              Wait Sleep waitTime=0.3
              If barrenoActual≟13
                MoveDirectionNode (selectedDirection=ZPlus toolParams=0.03, 0.04)
                  Until DISTANCE (allowActions=false deceleration=3 distanceNodeType=STOP) Distance=0.03; motionParameters(blendRadius=0)
                MoveJ speed 60 deg/s, acceleration 80 deg/s^2 (useActiveTCP=true) feature=Base
                  Waypoint Zona_der1: TCP in base x=-721.714 y=-174.597 z=506.289 mm, rx=2.1128 ry=-2.325 rz=0 rad; joints [0.057, -90.231, 90.368, -0.664, 90.292, 0.009] deg
                  Waypoint Posicion_Cero: TCP in base x=0.641 y=-324.742 z=1651.532 mm, rx=-0.0042 ry=-0.0154 rz=-3.0499 rad; joints [-0.001, -90.003, -0.001, -90, 0, 0.002] deg
                Call Quitar_Broca_Chida
                Call Poner_Broca
                MoveJ speed 60 deg/s, acceleration 80 deg/s^2 (useActiveTCP=true) feature=Base
                  Waypoint Posicion_Cero: TCP in base x=0.641 y=-324.742 z=1651.532 mm, rx=-0.0042 ry=-0.0154 rz=-3.0499 rad; joints [-0.001, -90.003, -0.001, -90, 0, 0.002] deg
                  Waypoint Zona_der1: TCP in base x=-721.714 y=-174.597 z=506.289 mm, rx=2.1128 ry=-2.325 rz=0 rad; joints [0.057, -90.231, 90.368, -0.664, 90.292, 0.009] deg
              ElseIf barrenoActual≟27
                MoveDirectionNode (selectedDirection=ZPlus toolParams=0.03, 0.04)
                  Until DISTANCE (allowActions=false deceleration=3 distanceNodeType=STOP) Distance=0.03; motionParameters(blendRadius=0)
                MoveJ speed 60 deg/s, acceleration 80 deg/s^2 (useActiveTCP=true) feature=Base
                  Waypoint Zona_der1: TCP in base x=-721.714 y=-174.597 z=506.289 mm, rx=2.1128 ry=-2.325 rz=0 rad; joints [0.057, -90.231, 90.368, -0.664, 90.292, 0.009] deg
                  Waypoint Posicion_Cero: TCP in base x=0.641 y=-324.742 z=1651.532 mm, rx=-0.0042 ry=-0.0154 rz=-3.0499 rad; joints [-0.001, -90.003, -0.001, -90, 0, 0.002] deg
                Call Quitar_Broca_Chida
                Set DigitalOutput pin=carrusel_home; digitalValue=1
                Wait Sleep waitTime=1
                Set DigitalOutput pin=carrusel_home; digitalValue=0
                Set ExpressionOutput pin=mensaje_mw10; expression=85
                Wait DigitalInput pin=Continuar_M30; digitalValue=1
                Wait Sleep waitTime=1
                Set ExpressionOutput pin=mensaje_mw10; expression=120
                Wait DigitalInput pin=Continuar_M30; digitalValue=1
                Wait Sleep waitTime=1
                Set DigitalOutput pin=carrusel_home; digitalValue=1
                Wait Sleep waitTime=1
                Set DigitalOutput pin=carrusel_home; digitalValue=0
                Set ExpressionOutput pin=mensaje_mw10; expression=90
                Wait DigitalInput pin=Continuar_M30; digitalValue=1
                Wait Sleep waitTime=1
                Call Poner_Broca
                broca := 217
                MoveJ speed 60 deg/s, acceleration 80 deg/s^2 (useActiveTCP=true) feature=Base
                  Waypoint Posicion_Cero: TCP in base x=0.641 y=-324.742 z=1651.532 mm, rx=-0.0042 ry=-0.0154 rz=-3.0499 rad; joints [-0.001, -90.003, -0.001, -90, 0, 0.002] deg
                  Waypoint Zona_der1: TCP in base x=-721.714 y=-174.597 z=506.289 mm, rx=2.1128 ry=-2.325 rz=0 rad; joints [0.057, -90.231, 90.368, -0.664, 90.292, 0.009] deg
                Set ExpressionOutput pin=mensaje_mw10; expression=95
                Wait DigitalInput pin=Continuar_M30; digitalValue=1
                Wait Sleep waitTime=1
                Set ExpressionOutput pin=mensaje_mw10; expression=150
                Wait DigitalInput pin=Continuar_M30; digitalValue=1
                Wait Sleep waitTime=1
              barrenoActual := barrenoActual+1
        Folder Linea 1 a 217
          broca := 217
          Folder Buje_inicial
            Buje_Inicial := L1B2
          Folder Buje_final
            Buje_Final := L1B1
          barrenosTotales := 27
          barrenoActual := 1
          Loop While (checkContinuously=false) expression=barrenoActual≤barrenosTotales
            MoveL speed 250 mm/s, acceleration 1200 mm/s^2 (useActiveTCP=true) feature=Base
              bajada_broca := p[0,0,0.018,0,0,0]
              internos := interpolate_pose(Buje_Inicial, Buje_Final, ((barrenoActual)-1)/((barrenosTotales)-1))
              Wait Sleep waitTime=2
              Folder Alturas
                If barrenoActual≟1 or barrenoActual≟3 or barrenoActual≟5 or barrenoActual≟7 or barrenoActual≟9 or barrenoActual≟11 or barrenoActual≟13 or barrenoActual≟15 or barrenoActual≟17 or barrenoActual≟19 or barrenoActual≟21 or barrenoActual≟23 or barrenoActual≟25 or barrenoActual≟27
                  Set ExpressionOutput pin=mensaje_mw10; expression=200
                  Wait DigitalInput pin=Continuar_M30; digitalValue=1
                  Wait Sleep waitTime=1
                  Set ExpressionOutput pin=mensaje_mw10; expression=150
                  Wait Sleep waitTime=1
                MoveJ speed 30 deg/s, acceleration 40 deg/s^2 (useActiveTCP=true) feature=Base
                  Waypoint Waypoint (Variable): variable=internos
                Wait Sleep waitTime=2
                If P1h[2]<P2h[2]
                  acomodo := (altura/(barrenosTotales-1))*(barrenoActual-1)
                  tcp := get_actual_tcp_pose()
                  offset_altura := p[tcp[0],tcp[1],((alta-0.0095)-(acomodo/1000)),tcp[3],tcp[4],tcp[5]]
                  MoveL speed 250 mm/s, acceleration 1200 mm/s^2 (useActiveTCP=true) feature=Base
                    Waypoint Waypoint (Variable): motionParameters(jointSpeed=1.047198 jointAcceleration=1.396263 cartesianSpeed=0.03 cartesianAcceleration=0.04); variable=offset_altura
                Else 
                  acomodo := (altura/(barrenosTotales-1))*(26-(barrenoActual-1))
                  tcp := get_actual_tcp_pose()
                  offset_altura := p[tcp[0],tcp[1],((alta-0.0095)-(acomodo/1000)),tcp[3],tcp[4],tcp[5]]
                  MoveL speed 250 mm/s, acceleration 1200 mm/s^2 (useActiveTCP=true) feature=Base
                    Waypoint Waypoint (Variable): motionParameters(jointSpeed=1.047198 jointAcceleration=1.396263 cartesianSpeed=0.03 cartesianAcceleration=0.04); variable=offset_altura
              Folder Freemove
                Wait Sleep waitTime=2
                Script: freedrive_mode()
                Wait Sleep waitTime=2.5
                Script: end_freedrive_mode()
              Wait Sleep waitTime=0.3
              Set DigitalOutput pin=config_out[1]; digitalValue=1
              Wait Sleep waitTime=1
              Wait Sleep waitTime=0.3
              Wait Sleep waitTime=0.3
              Wait Sleep waitTime=0.3
              Loop Counting (count=1) loopVariable(name=Loop_56)
                Poses_taladrado := pose_sub(get_actual_tcp_pose(), bajada_broca)
                Waypoint Waypoint (Variable): motionParameters(jointSpeed=1.047198 jointAcceleration=1.396263 cartesianSpeed=0.001 cartesianAcceleration=0.005); variable=Poses_taladrado
                If bajada_broca≟p[0,0,0.018,0,0,0]
                  num_barreno := str_cat("Barreno: ",barrenoActual)
                  tcp_actual := get_actual_tcp_pose()
                  X_actual := str_cat("     X: ",tcp_actual[0])
                  Y_actual := str_cat("     Y: ",tcp_actual[1])
                  pos_barreno := str_cat(X_actual,Y_actual)
                  Script: textmsg(num_barreno,pos_barreno)
                Poses_taladrado := pose_add(get_actual_tcp_pose(), bajada_broca)
                Waypoint Waypoint (Variable): motionParameters(jointSpeed=1.047198 jointAcceleration=1.396263 cartesianSpeed=0.01 cartesianAcceleration=0.01); variable=Poses_taladrado
                bajada_broca := pose_add(bajada_broca, p[0,0,0.018,0,0,0])
              MoveDirectionNode (selectedDirection=ZPlus toolParams=0.01, 0.01)
                Until DISTANCE (allowActions=false deceleration=3 distanceNodeType=STOP) Distance=0.05; motionParameters(blendRadius=0)
              MoveJ speed 30 deg/s, acceleration 40 deg/s^2 (useActiveTCP=true) feature=Base
                Waypoint Waypoint (Variable): variable=internos
              Wait Sleep waitTime=0.3
              Set DigitalOutput pin=config_out[1]; digitalValue=0
              Wait Sleep waitTime=0.3
              If barrenoActual≟13 or barrenoActual≟27
                MoveDirectionNode (selectedDirection=ZPlus toolParams=0.04, 0.03)
                  Until DISTANCE (allowActions=false deceleration=3 distanceNodeType=STOP) Distance=0.03; motionParameters(blendRadius=0)
                MoveJ speed 30 deg/s, acceleration 40 deg/s^2 (useActiveTCP=true) feature=Base
                  Waypoint Zona_der1: TCP in base x=-721.714 y=-174.597 z=506.289 mm, rx=2.1128 ry=-2.325 rz=0 rad; joints [0.057, -90.231, 90.368, -0.664, 90.292, 0.009] deg
                  Waypoint Posicion_Cero: TCP in base x=0.641 y=-324.742 z=1651.532 mm, rx=-0.0042 ry=-0.0154 rz=-3.0499 rad; joints [-0.001, -90.003, -0.001, -90, 0, 0.002] deg
                Call Quitar_Broca_Chida
                If barrenoActual≟13
                  Call Poner_Broca
                ElseIf barrenoActual≟27
                  Call Poner_Broca
                MoveJ speed 30 deg/s, acceleration 40 deg/s^2 (useActiveTCP=true) feature=Base
                  Waypoint Posicion_Cero: TCP in base x=0.641 y=-324.742 z=1651.532 mm, rx=-0.0042 ry=-0.0154 rz=-3.0499 rad; joints [-0.001, -90.003, -0.001, -90, 0, 0.002] deg
                  Waypoint Zona_der1: TCP in base x=-721.714 y=-174.597 z=506.289 mm, rx=2.1128 ry=-2.325 rz=0 rad; joints [0.057, -90.231, 90.368, -0.664, 90.292, 0.009] deg
              barrenoActual := barrenoActual+1
        Folder Linea 2 a 217
          broca := 217
          Folder Buje_inicial
            Buje_Inicial := L2B2
          Folder Buje_final
            Buje_Final := L2B1
          barrenosTotales := 27
          barrenoActual := 1
          Loop While (checkContinuously=false) expression=barrenoActual≤barrenosTotales
            MoveL speed 250 mm/s, acceleration 1200 mm/s^2 (useActiveTCP=true) feature=Base
              bajada_broca := p[0,0,0.018,0,0,0]
              internos := interpolate_pose(Buje_Inicial, Buje_Final, ((barrenoActual)-1)/((barrenosTotales)-1))
              Folder Alturas
                If barrenoActual≟1 or barrenoActual≟3 or barrenoActual≟5 or barrenoActual≟7 or barrenoActual≟9 or barrenoActual≟11 or barrenoActual≟13 or barrenoActual≟15 or barrenoActual≟17 or barrenoActual≟19 or barrenoActual≟21 or barrenoActual≟23 or barrenoActual≟25 or barrenoActual≟27
                  Set ExpressionOutput pin=mensaje_mw10; expression=200
                  Wait DigitalInput pin=Continuar_M30; digitalValue=1
                  Wait Sleep waitTime=1
                  Set ExpressionOutput pin=mensaje_mw10; expression=150
                  Wait Sleep waitTime=1
                MoveJ speed 30 deg/s, acceleration 40 deg/s^2 (useActiveTCP=true) feature=Base
                  Waypoint Waypoint (Variable): variable=internos
                Wait Sleep waitTime=2
                If P1h[2]<P2h[2]
                  acomodo := (altura/(barrenosTotales-1))*(barrenoActual-1)
                  tcp := get_actual_tcp_pose()
                  offset_altura := p[tcp[0],tcp[1],((alta-0.0095)-(acomodo/1000)),tcp[3],tcp[4],tcp[5]]
                  MoveL speed 250 mm/s, acceleration 1200 mm/s^2 (useActiveTCP=true) feature=Base
                    Waypoint Waypoint (Variable): motionParameters(jointSpeed=1.047198 jointAcceleration=1.396263 cartesianSpeed=0.03 cartesianAcceleration=0.04); variable=offset_altura
                Else 
                  acomodo := (altura/(barrenosTotales-1))*(26-(barrenoActual-1))
                  tcp := get_actual_tcp_pose()
                  offset_altura := p[tcp[0],tcp[1],((alta-0.0095)-(acomodo/1000)),tcp[3],tcp[4],tcp[5]]
                  MoveL speed 250 mm/s, acceleration 1200 mm/s^2 (useActiveTCP=true) feature=Base
                    Waypoint Waypoint (Variable): motionParameters(jointSpeed=1.047198 jointAcceleration=1.396263 cartesianSpeed=0.03 cartesianAcceleration=0.04); variable=offset_altura
              Folder Freemove
                Wait Sleep waitTime=2
                Script: freedrive_mode()
                Wait Sleep waitTime=2.5
                Script: end_freedrive_mode()
              Wait Sleep waitTime=0.3
              Set DigitalOutput pin=config_out[1]; digitalValue=1
              Wait Sleep waitTime=1
              Wait Sleep waitTime=0.3
              Wait Sleep waitTime=0.3
              Wait Sleep waitTime=0.3
              Loop Counting (count=1) loopVariable(name=Loop_58)
                Poses_taladrado := pose_sub(get_actual_tcp_pose(), bajada_broca)
                Waypoint Waypoint (Variable): motionParameters(jointSpeed=1.047198 jointAcceleration=1.396263 cartesianSpeed=0.001 cartesianAcceleration=0.005); variable=Poses_taladrado
                If bajada_broca≟p[0,0,0.018,0,0,0]
                  num_barreno := str_cat("Barreno: ",barrenoActual)
                  tcp_actual := get_actual_tcp_pose()
                  X_actual := str_cat("     X: ",tcp_actual[0])
                  Y_actual := str_cat("     Y: ",tcp_actual[1])
                  pos_barreno := str_cat(X_actual,Y_actual)
                  Script: textmsg(num_barreno,pos_barreno)
                Poses_taladrado := pose_add(get_actual_tcp_pose(), bajada_broca)
                Waypoint Waypoint (Variable): motionParameters(jointSpeed=1.047198 jointAcceleration=1.396263 cartesianSpeed=0.01 cartesianAcceleration=0.01); variable=Poses_taladrado
                bajada_broca := pose_add(bajada_broca, p[0,0,0.018,0,0,0])
              MoveDirectionNode (selectedDirection=ZPlus toolParams=0.01, 0.01)
                Until DISTANCE (allowActions=false deceleration=3 distanceNodeType=STOP) Distance=0.05; motionParameters(blendRadius=0)
              MoveJ speed 30 deg/s, acceleration 40 deg/s^2 (useActiveTCP=true) feature=Base
                Waypoint Waypoint (Variable): variable=internos
              Wait Sleep waitTime=0.3
              Set DigitalOutput pin=config_out[1]; digitalValue=0
              Wait Sleep waitTime=0.3
              If barrenoActual≟13
                MoveDirectionNode (selectedDirection=ZPlus toolParams=0.03, 0.04)
                  Until DISTANCE (allowActions=false deceleration=3 distanceNodeType=STOP) Distance=0.03; motionParameters(blendRadius=0)
                MoveJ speed 60 deg/s, acceleration 80 deg/s^2 (useActiveTCP=true) feature=Base
                  Waypoint Zona_der1: TCP in base x=-721.714 y=-174.597 z=506.289 mm, rx=2.1128 ry=-2.325 rz=0 rad; joints [0.057, -90.231, 90.368, -0.664, 90.292, 0.009] deg
                  Waypoint Posicion_Cero: TCP in base x=0.641 y=-324.742 z=1651.532 mm, rx=-0.0042 ry=-0.0154 rz=-3.0499 rad; joints [-0.001, -90.003, -0.001, -90, 0, 0.002] deg
                Call Quitar_Broca_Chida
                Call Poner_Broca
                MoveJ speed 60 deg/s, acceleration 80 deg/s^2 (useActiveTCP=true) feature=Base
                  Waypoint Posicion_Cero: TCP in base x=0.641 y=-324.742 z=1651.532 mm, rx=-0.0042 ry=-0.0154 rz=-3.0499 rad; joints [-0.001, -90.003, -0.001, -90, 0, 0.002] deg
                  Waypoint Zona_der1: TCP in base x=-721.714 y=-174.597 z=506.289 mm, rx=2.1128 ry=-2.325 rz=0 rad; joints [0.057, -90.231, 90.368, -0.664, 90.292, 0.009] deg
              ElseIf barrenoActual≟27
                MoveDirectionNode (selectedDirection=ZPlus toolParams=0.03, 0.04)
                  Until DISTANCE (allowActions=false deceleration=3 distanceNodeType=STOP) Distance=0.03; motionParameters(blendRadius=0)
                MoveJ speed 60 deg/s, acceleration 80 deg/s^2 (useActiveTCP=true) feature=Base
                  Waypoint Zona_der1: TCP in base x=-721.714 y=-174.597 z=506.289 mm, rx=2.1128 ry=-2.325 rz=0 rad; joints [0.057, -90.231, 90.368, -0.664, 90.292, 0.009] deg
                  Waypoint Posicion_Cero: TCP in base x=0.641 y=-324.742 z=1651.532 mm, rx=-0.0042 ry=-0.0154 rz=-3.0499 rad; joints [-0.001, -90.003, -0.001, -90, 0, 0.002] deg
                Call Quitar_Broca_Chida
                Set DigitalOutput pin=carrusel_home; digitalValue=1
                Wait Sleep waitTime=1
                Set DigitalOutput pin=carrusel_home; digitalValue=0
                Set ExpressionOutput pin=mensaje_mw10; expression=120
                Wait DigitalInput pin=Continuar_M30; digitalValue=1
                Wait Sleep waitTime=1
                Set ExpressionOutput pin=mensaje_mw10; expression=100
                Wait DigitalInput pin=Continuar_M30; digitalValue=1
                Wait Sleep waitTime=1
                MoveJ speed 60 deg/s, acceleration 80 deg/s^2 (useActiveTCP=true) feature=Base
                  Waypoint Traslacion_der: TCP in base x=174.612 y=-721.747 z=506.267 mm, rx=3.1383 ry=-0.1432 rz=0.0001 rad; joints [89.991, -90.247, 90.386, -0.667, 89.974, 0.014] deg
              barrenoActual := barrenoActual+1
      Set DigitalOutput pin=pos4_term_m612; digitalValue=1
      Wait Sleep waitTime=1
      Set DigitalOutput pin=pos4_term_m612; digitalValue=0
    SuppressedNode
      Folder GoNoGo
        SuppressedNode
          Wait Condition expression=mensaje_mw10≟35
        Set ExpressionOutput pin=mensaje_mw10; expression=55
        Wait DigitalInput pin=Continuar_M30; digitalValue=1
        Wait Sleep waitTime=1
        SuppressedNode
          Popup Message (haltProgram=false message=Colocar bujes 1645 inputType=Text)
        Set ExpressionOutput pin=mensaje_mw10; expression=60
        Wait DigitalInput pin=Continuar_M30; digitalValue=1
        Wait Sleep waitTime=1
        SuppressedNode
          Popup Message (haltProgram=false message=empezar gonogo inputType=Text)
        Folder Linea1_Buje1
          Xfin := ((0.09525*Xp)-(Xd)-(-0.0127*(1/m2)))*(-1)
          Yfin := ((-0.0127*Yp)-(Yd)+(0.09525*m1))*(-1)
          rotaciones := get_actual_tcp_pose()
          var_3 := rotaciones[3]
          var_4 := rotaciones[4]
          var_5 := rotaciones[5]
          If broca≟1645
            PosFinal := p[Xfin+0.00208915,Yfin+0.00208915,0.025,var_3,var_4,var_5]
          ElseIf broca≟1935
            PosFinal := p[Xfin+0.00245745,Yfin+0.00245745,0.025,var_3,var_4,var_5]
          ElseIf broca≟217
            PosFinal := p[Xfin+0.0027559,Yfin+0.0027559,0.025,var_3,var_4,var_5]
          Buje_Final := PosFinal
        MoveJ speed 60 deg/s, acceleration 80 deg/s^2 (useActiveTCP=true) feature=Base
          Waypoint Waypoint (Variable): variable=Buje_Final
        MoveL speed 60 mm/s, acceleration 80 mm/s^2 (useActiveTCP=true) feature=Base
          MoveDirectionNode (selectedDirection=ZMinus)
            Until DISTANCE (allowActions=false deceleration=3 distanceNodeType=STOP) Distance=0.03; motionParameters(blendRadius=0)
          MoveDirectionNode (selectedDirection=ZPlus)
            Until DISTANCE (allowActions=false deceleration=3 distanceNodeType=STOP) Distance=0.03; motionParameters(blendRadius=0)
          MoveDirectionNode (selectedDirection=XMinus)
            Until DISTANCE (allowActions=false deceleration=3 distanceNodeType=STOP) Distance=0.1; motionParameters(blendRadius=0)
        Folder Linea1_Buje2
          Xfin := ((0.75489*Xp)-(Xd)-(-0.01276*(1/m2)))*(-1)
          Yfin := ((-0.01276*Yp)-(Yd)+(0.75489*m1))*(-1)
          rotaciones := get_actual_tcp_pose()
          var_3 := rotaciones[3]
          var_4 := rotaciones[4]
          var_5 := rotaciones[5]
          If broca≟1645
            PosFinal := p[Xfin+0.00208915,Yfin+0.00208915,0.025,var_3,var_4,var_5]
          ElseIf broca≟1935
            PosFinal := p[Xfin+0.00245745,Yfin+0.00245745,0.025,var_3,var_4,var_5]
          ElseIf broca≟217
            PosFinal := p[Xfin+0.0027559,Yfin+0.0027559,0.025,var_3,var_4,var_5]
          Buje_Final := PosFinal
        MoveJ speed 60 deg/s, acceleration 80 deg/s^2 (useActiveTCP=true) feature=Base
          Waypoint Waypoint (Variable): variable=Buje_Final
        MoveL speed 60 mm/s, acceleration 80 mm/s^2 (useActiveTCP=true) feature=Base
          MoveDirectionNode (selectedDirection=ZMinus)
            Until DISTANCE (allowActions=false deceleration=3 distanceNodeType=STOP) Distance=0.03; motionParameters(blendRadius=0)
          MoveDirectionNode (selectedDirection=ZPlus)
            Until DISTANCE (allowActions=false deceleration=3 distanceNodeType=STOP) Distance=0.03; motionParameters(blendRadius=0)
        Folder Linea2_Buje2
          Xfin := ((0.75484*Xp)-(Xd)-(0.39312*(1/m2)))*(-1)
          Yfin := ((0.39312*Yp)-(Yd)+(0.75484*m1))*(-1)
          rotaciones := get_actual_tcp_pose()
          var_3 := rotaciones[3]
          var_4 := rotaciones[4]
          var_5 := rotaciones[5]
          If broca≟1645
            PosFinal := p[Xfin+0.00208915,Yfin+0.00208915,0.025,var_3,var_4,var_5]
          ElseIf broca≟1935
            PosFinal := p[Xfin+0.00245745,Yfin+0.00245745,0.025,var_3,var_4,var_5]
          ElseIf broca≟217
            PosFinal := p[Xfin+0.0027559,Yfin+0.0027559,0.025,var_3,var_4,var_5]
          Buje_Final := PosFinal
        MoveJ speed 60 deg/s, acceleration 80 deg/s^2 (useActiveTCP=true) feature=Base
          Waypoint Waypoint (Variable): variable=Buje_Final
        MoveL speed 60 mm/s, acceleration 80 mm/s^2 (useActiveTCP=true) feature=Base
          MoveDirectionNode (selectedDirection=ZMinus)
            Until DISTANCE (allowActions=false deceleration=3 distanceNodeType=STOP) Distance=0.03; motionParameters(blendRadius=0)
          MoveDirectionNode (selectedDirection=ZPlus)
            Until DISTANCE (allowActions=false deceleration=3 distanceNodeType=STOP) Distance=0.03; motionParameters(blendRadius=0)
          SuppressedNode
            MoveDirectionNode (selectedDirection=XMinus)
              Until DISTANCE (allowActions=false deceleration=3 distanceNodeType=STOP) Distance=0.1; motionParameters(blendRadius=0)
        Folder Linea2_Buje1
          Xfin := ((0.09525*Xp)-(Xd)-(0.3937*(1/m2)))*(-1)
          Yfin := ((0.3937*Yp)-(Yd)+(0.09525*m1))*(-1)
          rotaciones := get_actual_tcp_pose()
          var_3 := rotaciones[3]
          var_4 := rotaciones[4]
          var_5 := rotaciones[5]
          If broca≟1645
            PosFinal := p[Xfin+0.00208915,Yfin+0.00208915,0.025,var_3,var_4,var_5]
          ElseIf broca≟1935
            PosFinal := p[Xfin+0.00245745,Yfin+0.00245745,0.025,var_3,var_4,var_5]
          ElseIf broca≟217
            PosFinal := p[Xfin+0.0027559,Yfin+0.0027559,0.025,var_3,var_4,var_5]
          Buje_Final := PosFinal
        MoveJ speed 60 deg/s, acceleration 80 deg/s^2 (useActiveTCP=true) feature=Base
          Waypoint Waypoint (Variable): variable=Buje_Final
        MoveL speed 60 mm/s, acceleration 80 mm/s^2 (useActiveTCP=true) feature=Base
          MoveDirectionNode (selectedDirection=ZMinus)
            Until DISTANCE (allowActions=false deceleration=3 distanceNodeType=STOP) Distance=0.03; motionParameters(blendRadius=0)
          MoveDirectionNode (selectedDirection=ZPlus)
            Until DISTANCE (allowActions=false deceleration=3 distanceNodeType=STOP) Distance=0.03; motionParameters(blendRadius=0)
          SuppressedNode
            MoveDirectionNode (selectedDirection=XMinus)
              Until DISTANCE (allowActions=false deceleration=3 distanceNodeType=STOP) Distance=0.1; motionParameters(blendRadius=0)
        SuppressedNode
          Set ExpressionOutput pin=secuencia_mw11; expression=6
        SuppressedNode
          Set DigitalOutput pin=Msj_d_cobot_M31; digitalValue=1
        SuppressedNode
          Wait Sleep waitTime=1
        SuppressedNode
          Set DigitalOutput pin=Msj_d_cobot_M31; digitalValue=0
    SuppressedNode
      Set ExpressionOutput
    Folder Traslacion
      MoveJ speed 60 deg/s, acceleration 80 deg/s^2 (useActiveTCP=true) feature=Base
        Waypoint Traslacion_der: TCP in base x=174.612 y=-721.747 z=506.267 mm, rx=3.1383 ry=-0.1432 rz=0.0001 rad; joints [89.991, -90.247, 90.386, -0.667, 89.974, 0.014] deg
      Set ExpressionOutput pin=mensaje_mw10; expression=105
      Wait DigitalInput pin=Continuar_M30; digitalValue=1
      Wait Sleep waitTime=1
      Set ExpressionOutput pin=mensaje_mw10; expression=110
      Wait DigitalInput pin=Continuar_M30; digitalValue=1
      Wait Sleep waitTime=1
      Set DigitalOutput pin=postrnas_m187; digitalValue=1
      Wait Sleep waitTime=1
      Set DigitalOutput pin=Home_M20; digitalValue=1
      Wait Sleep waitTime=1
      Set DigitalOutput pin=Home_M20; digitalValue=0
      Set DigitalOutput pin=postrnas_m187; digitalValue=0
      Wait Sleep waitTime=10
    Folder Apagar
      Set ExpressionOutput pin=mensaje_mw10; expression=115
      Wait DigitalInput pin=Continuar_M30; digitalValue=1
      Wait Sleep waitTime=1
      MoveJ speed 60 deg/s, acceleration 80 deg/s^2 (useActiveTCP=true) feature=Base
        Waypoint Waypoint_8: TCP in base x=175.237 y=-168.919 z=168.903 mm, rx=3.0585 ry=-0.1387 rz=0.0062 rad; joints [90.001, -160.001, 154.893, -0.003, 90, 0.003] deg
        Waypoint Off_derecha: TCP in base x=175.178 y=-46.666 z=17.814 mm, rx=-1.9982 ry=0.0913 rz=0.0579 rad; joints [90, -90, 154.891, 0, 90, 0.001] deg
      Set ExpressionOutput pin=mensaje_mw10; expression=0
      Wait Sleep waitTime=1
      Wait DigitalInput pin=Continuar_M30; digitalValue=1
      Wait Sleep waitTime=1
      Popup Warning (haltProgram=true message=Apagar DAS inputType=Text)
  ElseIf Lado_Correr≟1
    Set ExpressionOutput pin=mensaje_mw10; expression=205
  ElseIf Lado_Correr≟0
    Set ExpressionOutput pin=mensaje_mw10; expression=205
  Else 
    Lado := False
    Set ExpressionOutput pin=mensaje_mw10; expression=205
    Popup Warning (haltProgram=true message=DAS no anclado inputType=Text)
SubProgram -> Poner_Broca
SubProgram -> Quitar_Broca_Chida
SubProgram -> Calibracion
SubProgram Poner_Broca (keepSynchronizedWithDisk=false)
  If Lado_Correr≟2
    Folder Poner_Broca
      Set DigitalOutput pin=ini_cambro_m289; digitalValue=0
      MoveJ speed 60 deg/s, acceleration 80 deg/s^2 (useActiveTCP=true) feature=Base
        Waypoint Precambio_der: TCP in base x=0.184 y=459.545 z=420.003 mm, rx=0.2788 ry=3.1256 rz=-0.0305 rad; joints [126.473, -59.389, -120.459, -180.773, -48.503, 0.207] deg
      MoveL speed 250 mm/s, acceleration 1200 mm/s^2 (useActiveTCP=true) feature=Base
        Waypoint Dejar_der: TCP in base x=0.169 y=459.556 z=61.15 mm, rx=0.2788 ry=3.1257 rz=-0.0305 rad; joints [126.442, -79.314, -149.852, -131.487, -48.653, 0.257] deg
      Set DigitalOutput pin=ini_cambro_m289; digitalValue=1
      Wait Sleep waitTime=3.8
      Set DigitalOutput pin=ini_cambro_m289; digitalValue=0
      Wait Sleep waitTime=0.5
      Wait DigitalInput pin=fciclocarr_m292; digitalValue=0
      Wait Sleep waitTime=0.5
      Script: freedrive_mode()
      Wait Sleep waitTime=2
      Script: end_freedrive_mode()
      MoveJ speed 60 deg/s, acceleration 80 deg/s^2 (useActiveTCP=true) feature=Base
        Waypoint Dejar_der: TCP in base x=0.169 y=459.556 z=61.15 mm, rx=0.2788 ry=3.1257 rz=-0.0305 rad; joints [126.442, -79.314, -149.852, -131.487, -48.653, 0.257] deg
      MoveL speed 250 mm/s, acceleration 1200 mm/s^2 (useActiveTCP=true) feature=Base
        Waypoint Precambio_der: TCP in base x=0.184 y=459.545 z=420.003 mm, rx=0.2788 ry=3.1256 rz=-0.0305 rad; joints [126.473, -59.389, -120.459, -180.773, -48.503, 0.207] deg
  ElseIf Lado_Correr≟1
    SuppressedNode
      Popup Message (haltProgram=false message=__ inputType=Text)
  ElseIf Lado_Correr≟0
    SuppressedNode
      Popup Message (haltProgram=false message=__ inputType=Text)
  Else 
    Lado := False
    Popup Warning (haltProgram=true message=DAS no anclado inputType=Text)
SubProgram Quitar_Broca_Chida (keepSynchronizedWithDisk=false)
  If Lado_Correr≟2
    Folder Quitar_Broca
      MoveJ speed 60 deg/s, acceleration 80 deg/s^2 (useActiveTCP=true) feature=Base
        Loop Counting (count=1) loopVariable(name=Loop_3)
          MoveL speed 250 mm/s, acceleration 1200 mm/s^2 (useActiveTCP=true) feature=Base
            MoveJ speed 60 deg/s, acceleration 80 deg/s^2 (useActiveTCP=true) feature=Base
              Waypoint Precambio_der: TCP in base x=0.184 y=459.545 z=420.003 mm, rx=0.2788 ry=3.1256 rz=-0.0305 rad; joints [126.473, -59.389, -120.459, -180.773, -48.503, 0.207] deg
            Waypoint Dejar_der: motionParameters(jointSpeed=1.047198 jointAcceleration=1.396263 cartesianSpeed=0.1 cartesianAcceleration=0.08); TCP in base x=0.169 y=459.556 z=61.15 mm, rx=0.2788 ry=3.1257 rz=-0.0305 rad; joints [126.442, -79.314, -149.852, -131.487, -48.653, 0.257] deg
            Wait Sleep waitTime=0.5
            Script: freedrive_mode()
            Wait Sleep waitTime=2
            Script: end_freedrive_mode()
            Set DigitalOutput pin=outputbroc_m291; digitalValue=1
            Wait Sleep waitTime=0.5
            Set DigitalOutput pin=outputbroc_m291; digitalValue=0
            Wait Sleep waitTime=0.5
            Wait DigitalInput pin=fciclocarr_m292; digitalValue=0
            Wait Sleep waitTime=0.5
            Script: freedrive_mode()
            Wait Sleep waitTime=2
            Script: end_freedrive_mode()
            Waypoint Precambio_der: TCP in base x=0.184 y=459.545 z=420.003 mm, rx=0.2788 ry=3.1256 rz=-0.0305 rad; joints [126.473, -59.389, -120.459, -180.773, -48.503, 0.207] deg
            Set DigitalOutput pin=avancarrusel_m7; digitalValue=1
            Wait Sleep waitTime=1.1
            Set DigitalOutput pin=avancarrusel_m7; digitalValue=0
  ElseIf Lado_Correr≟1
    SuppressedNode
      Popup Message (haltProgram=false message=_____ inputType=Text)
  ElseIf Lado_Correr≟0
    SuppressedNode
      Popup Message (haltProgram=false message=_____ inputType=Text)
  Else 
    Lado := False
    Popup Warning (haltProgram=true message=DAS no anclado inputType=Text)
SubProgram Calibracion (keepSynchronizedWithDisk=false)
  SuppressedNode
    Folder Offsets factor
      SuppressedNode
        broca := 1645
      L1B1x := ((0.09525254)/(0.09525))*(0.09525254)
      L1B1y := ((-0.01266698)/(-0.0127))*(-0.01266698)
      L1B2x := ((0.75576176)/(0.75565))*(0.75576176)
      L1B2y := ((-0.01269238)/(-0.0127))*(-0.01269238)
      L2B1x := ((0.09513062)/(0.09525))*(0.09525)
      L2B1y := ((0.39369238)/(0.3937))*(0.39369238)
      L2B2x := ((0.75565508)/(0.75565))*(0.75565508)
      L2B2y := ((0.39372032)/(0.3937))*(0.39372032)
  SuppressedNode
    Folder Offsets factor
      broca := 1645
      L1B1x := (((0.09525254)/(0.09525))*(0.09525254))*(1)
      L1B1y := (((-0.012)/(-0.0127))*(-0.012))*(1)
      L1B2x := (((0.74)/(0.75565))*(0.74))*(1.0003)
      L1B2y := (((-0.00986)/(-0.0127))*(-0.00986))*(1.0086956521739)
      L2B1x := ((0.09513062)/(0.09525))*(0.09525)
      L2B1y := ((0.39369238)/(0.3937))*(0.39369238)
      L2B2x := ((0.75565508)/(0.75565))*(0.75565508)
      L2B2y := ((0.39290032)/(0.3937))*(0.39290032)
  Folder Offsets factor
    broca := 1645
    L1B1x := ((0.09525))
    L1B1y := ((-0.0127))
    L1B2x := ((0.75565))
    L1B2y := (-0.0127)
    L2B1x := ((0.09525))
    L2B1y := ((0.3937))
    L2B2x := ((0.75565))
    L2B2y := ((0.3937))
  If Lado_Correr≟2
    Folder Subvariables
      muestras := 1
      muestrasTomadas := 0
      P1 := p[0,0,0,0,0,0]
      P2 := p[0,0,0,0,0,0]
      P3 := p[0,0,0,0,0,0]
      P4 := p[0,0,0,0,0,0]
      P1h := p[0,0,0,0,0,0]
      P2h := p[0,0,0,0,0,0]
      altura := 0
      rotaciones := p[0,0,0,0,0,0]
      PosFinal := p[0,0,0,0,0,0]
      m1 := 0
      m2 := 0
      b1 := 0
      b2 := 0
      Xd := 0
      Yd := 0
      Xp := 0
      Yp := 0
      Xfin := 0
      Yfin := 0
    Folder Calibracion
      MoveL speed 250 mm/s, acceleration 1200 mm/s^2 (useActiveTCP=true) feature=Base
        MoveDirectionNode (selectedDirection=ZPlus)
          Until DISTANCE (allowActions=false deceleration=3 distanceNodeType=STOP) Distance=0.1; motionParameters(blendRadius=0)
        MoveJ speed 60 deg/s, acceleration 80 deg/s^2 (useActiveTCP=true) feature=Base
          Waypoint Zona_der1: TCP in base x=-721.714 y=-174.597 z=506.289 mm, rx=2.1128 ry=-2.325 rz=0 rad; joints [0.057, -90.231, 90.368, -0.664, 90.292, 0.009] deg
        MoveL speed 250 mm/s, acceleration 1200 mm/s^2 (useActiveTCP=true) feature=Base
          MoveJ speed 60 deg/s, acceleration 80 deg/s^2 (useActiveTCP=true) feature=Base
            If pos_eje7_mw13≟1
              Waypoint Paso1_Der1: TCP in base x=-487.791 y=-375.841 z=78.447 mm, rx=2.1128 ry=-2.325 rz=0 rad; joints [28.02, -81.796, 129.534, -48.358, 118.161, -0.195] deg
            ElseIf pos_eje7_mw13≟2
              Waypoint Paso1_Der2: TCP in base x=-769.184 y=-406.838 z=70.614 mm, rx=2.1127 ry=-2.3251 rz=-0.0001 rad; joints [19.793, -62.703, 102.898, -40.77, 109.947, -0.104] deg; TCP offset x=0.151 y=-167.165 z=35.088 mm, rx=1.5784 ry=-0.0729 rz=0.0687 rad
          Folder P1
            Loop While (checkContinuously=false) expression=muestrasTomadas<muestras
              MoveJ speed 60 deg/s, acceleration 80 deg/s^2 (useActiveTCP=true) feature=Base
                If pos_eje7_mw13≟1
                  Waypoint Sacar1_der1: TCP in base x=-413.834 y=-368.954 z=39.26 mm, rx=2.1127 ry=-2.3249 rz=-0.0001 rad; joints [32.011, -82.38, 136.487, -54.749, 122.144, -0.231] deg; TCP offset x=0.151 y=-167.165 z=35.088 mm, rx=1.5784 ry=-0.0729 rz=0.0687 rad
                ElseIf pos_eje7_mw13≟2
                  Waypoint Sacar1_der2: TCP in base x=-425.6 y=-361.059 z=42.962 mm, rx=2.1125 ry=-2.3251 rz=0 rad; joints [30.253, -82.731, 136.294, -54.197, 120.397, -0.208] deg
              Wait Sleep waitTime=0.5
              MoveDirectionNode (selectedDirection=YPlus toolParams=0.0013, 2.0E-4)
                Until TOOL_CONTACT_DETECTION (allowActions=false retraction=0 decelerationAcceleration=9 decelerationAngularAcceleration=34.906585)
              Wait Sleep waitTime=2
              P1 := pose_add(get_actual_tcp_pose(), P1)
              muestrasTomadas := muestrasTomadas+1
            muestrasTomadas := 0
            var_1 := (P1[0])/muestras
            var_2 := (P1[1])/muestras
            rotaciones := get_actual_tcp_pose()
            var_3 := rotaciones[3]
            var_4 := rotaciones[4]
            var_5 := rotaciones[5]
            P1 := p[var_1,var_2,-0.37,var_3,var_4,var_5]
          Folder P1h
            Loop While (checkContinuously=false) expression=muestrasTomadas<muestras
              MoveDirectionNode (selectedDirection=ZPlus)
                Until DISTANCE (allowActions=false deceleration=3 distanceNodeType=STOP) Distance=0.03; motionParameters(blendRadius=0)
              MoveJ speed 60 deg/s, acceleration 80 deg/s^2 (useActiveTCP=true) feature=Base
                If pos_eje7_mw13≟1
                  Waypoint Sacar1h_der1: TCP in base x=-482.894 y=-364.215 z=62.588 mm, rx=2.1128 ry=-2.325 rz=-0.0001 rad; joints [27.034, -81.355, 131.405, -50.661, 117.17, -0.179] deg
                ElseIf pos_eje7_mw13≟2
                  Waypoint Sacar1h_der2: TCP in base x=-495.382 y=-357.99 z=85.829 mm, rx=-2.1127 ry=2.3251 rz=0 rad; joints [25.656, -83.152, 130.077, -47.525, 115.803, -0.171] deg
              Wait Sleep waitTime=0.5
              MoveDirectionNode (selectedDirection=ZMinus)
                Until DISTANCE (allowActions=false deceleration=3 distanceNodeType=STOP) Distance=0.02; motionParameters(blendRadius=0)
              MoveDirectionNode (selectedDirection=ZMinus toolParams=0.0013, 2.0E-4)
                Until TOOL_CONTACT_DETECTION (allowActions=false retraction=0 decelerationAcceleration=9 decelerationAngularAcceleration=34.906585)
              Wait Sleep waitTime=2
              P1h := pose_add(get_actual_tcp_pose(), P1h)
              muestrasTomadas := muestrasTomadas+1
            muestrasTomadas := 0
            var_1 := (P1h[0])/muestras
            var_2 := (P1h[1])/muestras
            var_9 := (P1h[2])/muestras
            rotaciones := get_actual_tcp_pose()
            var_3 := rotaciones[3]
            var_4 := rotaciones[4]
            var_5 := rotaciones[5]
            P1h := p[var_1,var_2,var_9,var_3,var_4,var_5]
          MoveJ speed 60 deg/s, acceleration 80 deg/s^2 (useActiveTCP=true) feature=Base
            If pos_eje7_mw13≟1
              Waypoint Paso1_Der1: TCP in base x=-487.791 y=-375.841 z=78.447 mm, rx=2.1128 ry=-2.325 rz=0 rad; joints [28.02, -81.796, 129.534, -48.358, 118.161, -0.195] deg
              Waypoint Waypoint_9: TCP in base x=-607.44 y=-375.849 z=78.449 mm, rx=2.1127 ry=-2.325 rz=0.0001 rad; joints [22.399, -74.638, 120.095, -46.044, 112.542, -0.125] deg
            ElseIf pos_eje7_mw13≟2
              Waypoint Paso1_Der2: TCP in base x=-769.184 y=-406.838 z=70.614 mm, rx=2.1127 ry=-2.3251 rz=-0.0001 rad; joints [19.793, -62.703, 102.898, -40.77, 109.947, -0.104] deg; TCP offset x=0.151 y=-167.165 z=35.088 mm, rx=1.5784 ry=-0.0729 rz=0.0687 rad
          Folder P2
            Loop While (checkContinuously=false) expression=muestrasTomadas<muestras
              MoveJ speed 60 deg/s, acceleration 80 deg/s^2 (useActiveTCP=true) feature=Base
                If pos_eje7_mw13≟1
                  Waypoint Sacar2_der1: TCP in base x=-1163.96 y=-371.854 z=42.187 mm, rx=2.1127 ry=-2.325 rz=0.0001 rad; joints [10.901, -31.924, 49.952, -18.571, 101.103, -0.022] deg; TCP offset x=0.151 y=-167.165 z=35.088 mm, rx=1.5784 ry=-0.0729 rz=0.0687 rad
                ElseIf pos_eje7_mw13≟2
                  Waypoint Sacar2_der2: TCP in base x=-1175.947 y=-378.923 z=43.215 mm, rx=2.1125 ry=-2.3252 rz=-0.0001 rad; joints [11.151, -30.302, 46.666, -16.916, 101.365, -0.031] deg
              Wait Sleep waitTime=0.5
              MoveDirectionNode (selectedDirection=YPlus toolParams=0.0013, 2.0E-4)
                Until TOOL_CONTACT_DETECTION (allowActions=false retraction=0 decelerationAcceleration=9 decelerationAngularAcceleration=34.906585)
              Wait Sleep waitTime=2
              P2 := pose_add(get_actual_tcp_pose(), P2)
              muestrasTomadas := muestrasTomadas+1
            muestrasTomadas := 0
            var_1 := (P2[0])/muestras
            var_2 := (P2[1])/muestras
            rotaciones := get_actual_tcp_pose()
            var_3 := rotaciones[3]
            var_4 := rotaciones[4]
            var_5 := rotaciones[5]
            P2 := p[var_1,var_2,-0.37,var_3,var_4,var_5]
          Folder P2h
            Loop While (checkContinuously=false) expression=muestrasTomadas<muestras
              MoveJ speed 60 deg/s, acceleration 80 deg/s^2 (useActiveTCP=true) feature=Base
                If pos_eje7_mw13≟1
                  Waypoint Waypoint_11: TCP in base x=-1163.976 y=-371.873 z=73.926 mm, rx=2.1127 ry=-2.325 rz=0.0001 rad; joints [10.901, -33.06, 48.835, -16.323, 101.108, -0.023] deg
                  Waypoint Waypoint_10: TCP in base x=-1131.947 y=-365.226 z=69.177 mm, rx=2.1126 ry=-2.3249 rz=0.0001 rad; joints [10.876, -36.582, 56.111, -20.08, 101.072, -0.019] deg
                ElseIf pos_eje7_mw13≟2
                  Waypoint Paso1_Der2: TCP in base x=-769.184 y=-406.838 z=70.614 mm, rx=2.1127 ry=-2.3251 rz=-0.0001 rad; joints [19.793, -62.703, 102.898, -40.77, 109.947, -0.104] deg; TCP offset x=0.151 y=-167.165 z=35.088 mm, rx=1.5784 ry=-0.0729 rz=0.0687 rad
                  Waypoint Sacar2h_der2: TCP in base x=-1152.872 y=-362.091 z=46.763 mm, rx=2.1127 ry=-2.325 rz=-0.0002 rad; joints [10.494, -33.687, 52.91, -19.778, 100.692, -0.024] deg; TCP offset x=0.151 y=-167.165 z=35.088 mm, rx=1.5784 ry=-0.0729 rz=0.0687 rad
              Wait Sleep waitTime=0.5
              MoveDirectionNode (selectedDirection=ZMinus toolParams=0.0013, 2.0E-4)
                Until TOOL_CONTACT_DETECTION (allowActions=false retraction=0 decelerationAcceleration=9 decelerationAngularAcceleration=34.906585)
              Wait Sleep waitTime=2
              P2h := pose_add(get_actual_tcp_pose(), P2h)
              muestrasTomadas := muestrasTomadas+1
            muestrasTomadas := 0
            var_1 := (P2h[0])/muestras
            var_2 := (P2h[1])/muestras
            var_9 := (P2h[2])/muestras
            rotaciones := get_actual_tcp_pose()
            var_3 := rotaciones[3]
            var_4 := rotaciones[4]
            var_5 := rotaciones[5]
            P2h := p[var_1,var_2,var_9,var_3,var_4,var_5]
          MoveJ speed 60 deg/s, acceleration 80 deg/s^2 (useActiveTCP=true) feature=Base
            If pos_eje7_mw13≟1
              Waypoint Waypoint_9: TCP in base x=-607.44 y=-375.849 z=78.449 mm, rx=2.1127 ry=-2.325 rz=0.0001 rad; joints [22.399, -74.638, 120.095, -46.044, 112.542, -0.125] deg
              Waypoint Paso1_Der1: TCP in base x=-487.791 y=-375.841 z=78.447 mm, rx=2.1128 ry=-2.325 rz=0 rad; joints [28.02, -81.796, 129.534, -48.358, 118.161, -0.195] deg
            ElseIf pos_eje7_mw13≟2
              Waypoint Paso1_Der2: TCP in base x=-769.184 y=-406.838 z=70.614 mm, rx=2.1127 ry=-2.3251 rz=-0.0001 rad; joints [19.793, -62.703, 102.898, -40.77, 109.947, -0.104] deg; TCP offset x=0.151 y=-167.165 z=35.088 mm, rx=1.5784 ry=-0.0729 rz=0.0687 rad
          Folder m1
            var_1 := (P1[0])
            var_2 := (P1[1])
            var_3 := (P2[0])
            var_4 := (P2[1])
            m1 := (var_4-var_2)/(var_3-var_1)
          Folder b1
            b1 := ((m1*var_1)-var_2)*(-1)
          MoveJ speed 60 deg/s, acceleration 80 deg/s^2 (useActiveTCP=true) feature=Base
            If pos_eje7_mw13≟1
              Waypoint Paso2_der1: TCP in base x=-429.675 y=-212.098 z=78.415 mm, rx=-2.1128 ry=2.325 rz=-0.0001 rad; joints [7.483, -97.666, 145.53, -48.399, 97.629, 0.008] deg; TCP offset x=0.151 y=-167.165 z=35.088 mm, rx=1.5784 ry=-0.0729 rz=0.0687 rad
            ElseIf pos_eje7_mw13≟2
              Waypoint Paso2_der2: TCP in base x=-416.303 y=-231.102 z=83.617 mm, rx=-2.1041 ry=2.3159 rz=-0.0179 rad; joints [11.332, -97.876, 144.551, -46.23, 101.494, 0.16] deg
          Folder P3
            Loop While (checkContinuously=false) expression=muestrasTomadas<muestras
              MoveJ speed 60 deg/s, acceleration 80 deg/s^2 (useActiveTCP=true) feature=Base
                If pos_eje7_mw13≟1
                  Waypoint Sacar3_der1: TCP in base x=-387.228 y=-86.478 z=43.603 mm, rx=2.1127 ry=-2.325 rz=-0.0001 rad; joints [-23.854, -108.598, 157.726, -49.681, 66.3, 0.301] deg
                ElseIf pos_eje7_mw13≟2
                  Waypoint Sacar3_der2: TCP in base x=-404.091 y=-76.521 z=43.707 mm, rx=-2.1022 ry=2.3133 rz=-0.0222 rad; joints [-24.089, -105.407, 155.567, -49.384, 66.061, -0.241] deg
              Wait Sleep waitTime=0.5
              MoveDirectionNode (selectedDirection=XPlus toolParams=0.0013, 2.0E-4)
                Until TOOL_CONTACT_DETECTION (allowActions=false retraction=0 decelerationAcceleration=9 decelerationAngularAcceleration=34.906585)
              Wait Sleep waitTime=2
              P3 := pose_add(get_actual_tcp_pose(), P3)
              muestrasTomadas := muestrasTomadas+1
            muestrasTomadas := 0
            var_1 := (P3[0])/muestras
            var_2 := (P3[1])/muestras
            rotaciones := get_actual_tcp_pose()
            var_3 := rotaciones[3]
            var_4 := rotaciones[4]
            var_5 := rotaciones[5]
            P3 := p[var_1,var_2,-0.37,var_3,var_4,var_5]
          MoveJ speed 60 deg/s, acceleration 80 deg/s^2 (useActiveTCP=true) feature=Base
            If pos_eje7_mw13≟1
              Waypoint Paso2_der1: TCP in base x=-429.675 y=-212.098 z=78.415 mm, rx=-2.1128 ry=2.325 rz=-0.0001 rad; joints [7.483, -97.666, 145.53, -48.399, 97.629, 0.008] deg
            ElseIf pos_eje7_mw13≟2
              Waypoint Paso2_der2: TCP in base x=-416.303 y=-231.102 z=83.617 mm, rx=-2.1041 ry=2.3159 rz=-0.0179 rad; joints [11.332, -97.876, 144.551, -46.23, 101.494, 0.16] deg
          Folder P4
            Loop While (checkContinuously=false) expression=muestrasTomadas<muestras
              MoveJ speed 60 deg/s, acceleration 80 deg/s^2 (useActiveTCP=true) feature=Base
                If pos_eje7_mw13≟1
                  Waypoint Sacar4_der1: TCP in base x=-385.951 y=-340.145 z=45.401 mm, rx=-2.1128 ry=2.325 rz=0 rad; joints [30.536, -86.673, 140.479, -54.431, 120.672, -0.215] deg
                ElseIf pos_eje7_mw13≟2
                  Waypoint Sacar4_der2: TCP in base x=-399.044 y=-315.798 z=44.221 mm, rx=-2.104 ry=2.316 rz=-0.0179 rad; joints [26.036, -87.615, 141.274, -53.174, 116.188, 0.313] deg
              Wait Sleep waitTime=0.5
              MoveDirectionNode (selectedDirection=XPlus toolParams=0.0013, 2.0E-4)
                Until TOOL_CONTACT_DETECTION (allowActions=false retraction=0 decelerationAcceleration=9 decelerationAngularAcceleration=34.906585)
              Wait Sleep waitTime=2
              P4 := pose_add(get_actual_tcp_pose(), P4)
              muestrasTomadas := muestrasTomadas+1
            muestrasTomadas := 0
            var_1 := (P4[0])/muestras
            var_2 := (P4[1])/muestras
            rotaciones := get_actual_tcp_pose()
            var_3 := rotaciones[3]
            var_4 := rotaciones[4]
            var_5 := rotaciones[5]
            P4 := p[var_1,var_2,-0.37,var_3,var_4,var_5]
          MoveJ speed 60 deg/s, acceleration 80 deg/s^2 (useActiveTCP=true) feature=Base
            If pos_eje7_mw13≟1
              Waypoint Paso2_der1: TCP in base x=-429.675 y=-212.098 z=78.415 mm, rx=-2.1128 ry=2.325 rz=-0.0001 rad; joints [7.483, -97.666, 145.53, -48.399, 97.629, 0.008] deg
            ElseIf pos_eje7_mw13≟2
              Waypoint Paso2_der2: TCP in base x=-416.303 y=-231.102 z=83.617 mm, rx=-2.1041 ry=2.3159 rz=-0.0179 rad; joints [11.332, -97.876, 144.551, -46.23, 101.494, 0.16] deg
          Folder m2
            var_1 := (P3[0])
            var_2 := (P3[1])
            var_3 := (P4[0])
            var_4 := (P4[1])
            m2 := (var_4-var_2)/(var_3-var_1)
          Folder b2
            b2 := ((m2*var_1)-var_2)*(-1)
          Folder Xd y Yd
            Xd := (b2-b1)/(m1-m2)
            Yd := (m1*Xd)+b1
          SuppressedNode
            Folder Zp
              Zp := (pow(((P1h[0])-(P2h[0])),2))+(pow(((P1h[1])-(P2h[1])),2))
              Zp := (Zp)/(pow((P1h[2]-P2h[2]),2)+Zp)
              Zp := sqrt(Zp)
          Folder Xp y Yp
            Xp := ((1)/(sqrt((m1*m1)+1)))*(1)
            Yp := ((m2)/(sqrt((m2*m2)+1)))*(1)
          Folder Origen
            Xfin := ((0*Xp)-(Xd)-(0*(1/m2)))*(-1)
            Yfin := ((0*Yp)-(Yd)+(0*m1))*(-1)
            rotaciones := get_actual_tcp_pose()
            var_3 := rotaciones[3]
            var_4 := rotaciones[4]
            var_5 := rotaciones[5]
            If broca≟1645
              PosFinal := p[Xfin+0.00208915,Yfin+0.00208915,0.065,var_3,var_4,var_5]
            ElseIf broca≟1935
              PosFinal := p[Xfin+0.00245745,Yfin+0.00245745,0.065,var_3,var_4,var_5]
            ElseIf broca≟217
              PosFinal := p[Xfin+0.0027559,Yfin+0.0027559,0.065,var_3,var_4,var_5]
            origen := PosFinal
          Folder Linea1_Buje1
            Xfin := (((L1B1x)*Xp)-(Xd)-((L1B1y)*(1/m2)))*(-1)
            Yfin := (((L1B1y)*Yp)-(Yd)+((L1B1x)*m1))*(-1)
            rotaciones := get_actual_tcp_pose()
            var_3 := rotaciones[3]
            var_4 := rotaciones[4]
            var_5 := rotaciones[5]
            If broca≟1645
              PosFinal := p[(Xfin+0.00208915)*1000,(Yfin+0.00208915)*1000,0.065,var_3,var_4,var_5]
            ElseIf broca≟1935
              PosFinal := p[Xfin+0.00245745,Yfin+0.00245745,0.065,var_3,var_4,var_5]
            ElseIf broca≟217
              PosFinal := p[Xfin+0.0027559,Yfin+0.0027559,0.065,var_3,var_4,var_5]
            Linea1_Buje1 := PosFinal
          Folder Linea1_Buje27
            Xfin := (((L1B2x)*Xp)-(Xd)-((L1B2y)*(1/m2)))*(-1)
            Yfin := (((L1B2y)*Yp)-(Yd)+((L1B2x)*m1))*(-1)
            rotaciones := get_actual_tcp_pose()
            var_3 := rotaciones[3]
            var_4 := rotaciones[4]
            var_5 := rotaciones[5]
            If broca≟1645
              PosFinal := p[(Xfin+0.00208915)*1000,(Yfin+0.00208915)*1000,0.065,var_3,var_4,var_5]
            ElseIf broca≟1935
              PosFinal := p[Xfin+0.00245745,Yfin+0.00245745,0.065,var_3,var_4,var_5]
            ElseIf broca≟217
              PosFinal := p[Xfin+0.0027559,Yfin+0.0027559,0.065,var_3,var_4,var_5]
            Linea1_Buje27 := PosFinal
          Folder Linea2_Buje1
            Xfin := (((L2B1x)*Xp)-(Xd)-((L2B1y)*(1/m2)))*(-1)
            Yfin := (((L2B1y)*Yp)-(Yd)+((L2B1x)*m1))*(-1)
            rotaciones := get_actual_tcp_pose()
            var_3 := rotaciones[3]
            var_4 := rotaciones[4]
            var_5 := rotaciones[5]
            If broca≟1645
              PosFinal := p[(Xfin+0.00208915)*1000,(Yfin+0.00208915)*1000,0.065,var_3,var_4,var_5]
            ElseIf broca≟1935
              PosFinal := p[Xfin+0.00245745,Yfin+0.00245745,0.065,var_3,var_4,var_5]
            ElseIf broca≟217
              PosFinal := p[Xfin+0.0027559,Yfin+0.0027559,0.065,var_3,var_4,var_5]
            Linea2_Buje1 := PosFinal
          Folder Linea2_Buje27
            Xfin := (((L2B2x)*Xp)-(Xd)-((L2B2y)*(1/m2)))*(-1)
            Yfin := (((L2B2y)*Yp)-(Yd)+((L2B2x)*m1))*(-1)
            rotaciones := get_actual_tcp_pose()
            var_3 := rotaciones[3]
            var_4 := rotaciones[4]
            var_5 := rotaciones[5]
            If broca≟1645
              PosFinal := p[(Xfin+0.00208915)*1000,(Yfin+0.00208915)*1000,0.065,var_3,var_4,var_5]
            ElseIf broca≟1935
              PosFinal := p[Xfin+0.00245745,Yfin+0.00245745,0.065,var_3,var_4,var_5]
            ElseIf broca≟217
              PosFinal := p[Xfin+0.0027559,Yfin+0.0027559,0.065,var_3,var_4,var_5]
            Linea2_Buje27 := PosFinal
          Folder Altura
            If P1h[2]<P2h[2]
              altura := (P2h[2]-P1h[2])*1000
              alta := (P2h[2])
            Else 
              altura := (P1h[2]-P2h[2])*1000
              alta := (P1h[2])
          MoveDirectionNode (selectedDirection=ZPlus)
            Until DISTANCE (allowActions=false deceleration=3 distanceNodeType=STOP) Distance=0.1; motionParameters(blendRadius=0)
          MoveJ speed 60 deg/s, acceleration 80 deg/s^2 (useActiveTCP=true) feature=Base
            Waypoint Zona_der1: TCP in base x=-721.714 y=-174.597 z=506.289 mm, rx=2.1128 ry=-2.325 rz=0 rad; joints [0.057, -90.231, 90.368, -0.664, 90.292, 0.009] deg
  ElseIf Lado_Correr≟1
    SuppressedNode
      Popup Message (haltProgram=false message=__ inputType=Text)
  ElseIf Lado_Correr≟0
    SuppressedNode
      Popup Message (haltProgram=false message=__ inputType=Text)
  Else 
    Lado := False
    Popup Warning (haltProgram=true message=DAS no anclado inputType=Text)
